{attribute addProperty BoxType ""}
{attribute addProperty Id "defaultSyncUnitTasks_5F8F1DD713016.250"}
{attribute addProperty CRC "3153825492"}
{attribute addProperty SizeInBites "130"}
{attribute addProperty SizeInBytes "16.25"}
TYPE SyncUnits_BBFB8ED4 :
STRUCT
	{attribute addProperty Name "default"}
	default : SyncUnitTasks_5F8F1DD7;
END_STRUCT
END_TYPE

(* stored: Version 1.2.0.0, ProductVersion 3.1.4024.9
   DUT SyncUnits_BBFB8ED4: Id {0a507494-2b07-4882-af40-9358ec1ad827} *)
